// TIA Portal project "Ejercicio2" (V15.1)

(* hardware
DEVICE "HMI_1"  KTP700 Basic PN
   slot 0: "HMI_1"  KTP700 Basic PN  6AV2 123-2GB03-0AX0  15.1.0.0
   slot 1: "HMI_RT_1"  KTP700 Basic PN  6AV2 123-2GB03-0AX0  15.1.0.0
   slot 5: "HMI_1.IE_CP_1"  PROFINET Interface  15.0.1.0
      slot 1: "Interfaz PROFINET_1"  PROFINET Interface
         slot 1: "Port_1"  Port
DEVICE "S7-1200 station_1"  S7-1200 Station
   slot 0: "Rack_0"  S7-1200 Rack  Rack  V1.0
   slot 1: "PLC_1"  CPU 1215C AC/DC/Rly  6ES7 215-1BG40-0XB0  V4.2
*)

// ===== PLC "PLC_1"  CPU 1215C AC/DC/Rly =====

VAR_GLOBAL   // PLC tag table "Tabla de variables estándar"
   "System_Byte" AT %MB8191 : Byte;
   "FirstScan" AT %M8191.0 : Bool;
   "DiagStatusUpdate" AT %M8191.1 : Bool;
   "AlwaysTRUE" AT %M8191.2 : Bool;
   "AlwaysFALSE" AT %M8191.3 : Bool;
   "System_Byte(1)" AT %MB1 : Byte;
   "Clock_Byte" AT %MB100 : Byte;
   "Clock_10Hz" AT %M100.0 : Bool;
   "Clock_5Hz" AT %M100.1 : Bool;
   "Clock_2.5Hz" AT %M100.2 : Bool;
   "Clock_2Hz" AT %M100.3 : Bool;
   "Clock_1.25Hz" AT %M100.4 : Bool;
   "Clock_1Hz" AT %M100.5 : Bool;
   "Clock_0.625Hz" AT %M100.6 : Bool;
   "Clock_0.5Hz" AT %M100.7 : Bool;
   "Zona 1" AT %M0.0 : Bool;
   "Zona 2" AT %M0.1 : Bool;
   "Alarma ON/OFF" AT %M0.2 : Bool;
   "Alarma manual" AT %M0.3 : Bool;
   "LED sistema de alarma" AT %M10.0 : Bool;
   "Sirenea de alarma" AT %M10.1 : Bool;
   "Señal de alerta baja" AT %M10.2 : Bool;
   "Activar relé" AT %M10.3 : Bool;
   "Estado Alarma" AT %M1.0 : Bool;
   "Estado Sirena" AT %M1.1 : Bool;
END_VAR

// folder: System blocks/Program resources

DATA_BLOCK "Temporizador90s"   // DB1
{ S7_Optimized_Access := 'TRUE' }
AUTHOR : Simatic
FAMILY : IEC
NAME : IEC_TMR
VERSION : 1.0
// stored: InstanceOfName IEC_TIMER
"IEC_TIMER"
BEGIN
END_DATA_BLOCK

DATA_BLOCK "Temporizador60s"   // DB2
{ S7_Optimized_Access := 'TRUE' }
AUTHOR : Simatic
FAMILY : IEC
NAME : IEC_TMR
VERSION : 1.0
// stored: InstanceOfName IEC_TIMER
"IEC_TIMER"
BEGIN
END_DATA_BLOCK

// folder: (top level)

ORGANIZATION_BLOCK "Main"   // OB1, LAD, ProgramCycle
TITLE = "Main Program Sweep (Cycle)"
{ S7_Optimized_Access := 'TRUE' }
VERSION : 0.1
   VAR_INPUT
      Initial_Call : Bool;   // Initial call of this OB
      Remanence : Bool;   // =True, if remanent data are available
   END_VAR
   VAR_TEMP   // added for the SCL form of the ladder/FBD networks
      _w1 : Bool;
   END_VAR
BEGIN

REGION Network 1: Encendido si está activado y parpadeante desactivado si zonas 1 y 2 abiertas
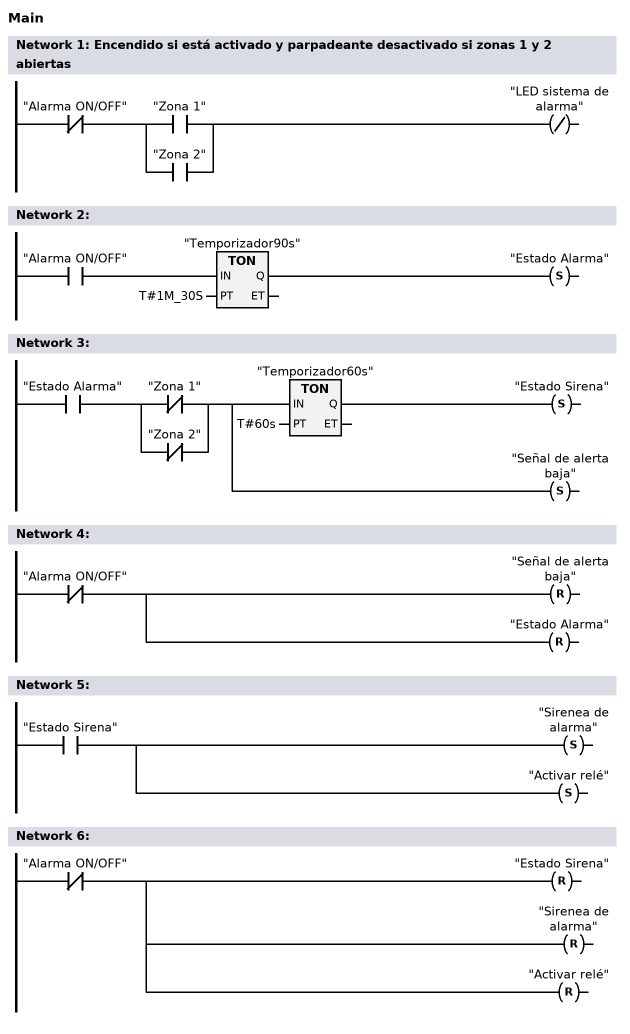
   RUNG wire#powerrail
      I_Contact( "Alarma ON/OFF" )
      wire#w1
      Contact( "Zona 1" )
      wire#w2
      I_Coil( "LED sistema de alarma" )
   END_RUNG
   RUNG wire#w1
      Contact( "Zona 2" )
   END_RUNG wire#w2
   // the same network as SCL:
   "LED sistema de alarma" := NOT (NOT "Alarma ON/OFF" AND ("Zona 1" OR "Zona 2"));
END_REGION

REGION Network 2
   "Temporizador90s".TON(IN := "Alarma ON/OFF", PT := T#1M_30S);
   IF "Temporizador90s".Q THEN "Estado Alarma" := TRUE; END_IF;
END_REGION

REGION Network 3
   #_w1 := "Estado Alarma" AND (NOT "Zona 1" OR NOT "Zona 2");
   "Temporizador60s".TON(IN := #_w1, PT := T#60s);
   IF "Temporizador60s".Q THEN "Estado Sirena" := TRUE; END_IF;
   IF #_w1 THEN "Señal de alerta baja" := TRUE; END_IF;
END_REGION

REGION Network 4
   RUNG wire#powerrail
      I_Contact( "Alarma ON/OFF" )
      wire#w1
      R_Coil( "Señal de alerta baja" )
   END_RUNG
   RUNG wire#w1
      R_Coil( "Estado Alarma" )
   END_RUNG
   // the same network as SCL:
   IF NOT "Alarma ON/OFF" THEN
       "Señal de alerta baja" := FALSE;
       "Estado Alarma" := FALSE;
   END_IF;
END_REGION

REGION Network 5
   RUNG wire#powerrail
      Contact( "Estado Sirena" )
      wire#w1
      S_Coil( "Sirenea de alarma" )
   END_RUNG
   RUNG wire#w1
      S_Coil( "Activar relé" )
   END_RUNG
   // the same network as SCL:
   IF "Estado Sirena" THEN
       "Sirenea de alarma" := TRUE;
       "Activar relé" := TRUE;
   END_IF;
END_REGION

REGION Network 6
   RUNG wire#powerrail
      I_Contact( "Alarma ON/OFF" )
      wire#w1
      R_Coil( "Estado Sirena" )
   END_RUNG
   RUNG wire#w1
      R_Coil( "Sirenea de alarma" )
   END_RUNG
   RUNG wire#w1
      R_Coil( "Activar relé" )
   END_RUNG
   // the same network as SCL:
   IF NOT "Alarma ON/OFF" THEN
       "Estado Sirena" := FALSE;
       "Sirenea de alarma" := FALSE;
       "Activar relé" := FALSE;
   END_IF;
END_REGION
END_ORGANIZATION_BLOCK

(* ===== HMI "HMI_RT_1" =====
system functions are stored by id; their names below are inferred from use
connection "HMI_Conexión_1": ETHERNET, SMART_S7_1200_OMS

HMI tags "Tabla de variables estándar"
   "Número_imagen_variable" : UInt, internal
   "Alarma ON/OFF" : Bool = PLC "Alarma ON/OFF" AT %M0.2, 1 s
   "Estado Alarma" : Bool = PLC "Estado Alarma" AT %M1.0, 1 s
   "Señal de alerta baja" : Bool = PLC "Señal de alerta baja" AT %M10.2, 1 s
   "Activar relé" : Bool = PLC "Activar relé" AT %M10.3, 1 s
   "LED sistema de alarma" : Bool = PLC "LED sistema de alarma" AT %M10.0, 1 s
   "Sirenea de alarma" : Bool = PLC "Sirenea de alarma" AT %M10.1, 1 s
   "Temporizador60s_ET" : Time = PLC Temporizador60s.ET, 1 s
   "Temporizador90s_ET" : Time = PLC Temporizador90s.ET, 1 s
   "Estado Sirena" : Bool = PLC "Estado Sirena" AT %M1.1, 1 s

text list "Nombre_imagen_lista_texto": 1 'Imagen raíz'

Template "Plantilla_1" 800x480
   Button "Salir" at 714,429 size 71x50; TextOff 'Salir'; PictureOff "ExitRuntime_KTP700_Basic_PN_TR"; PictureOn "ExitRuntime_KTP700_Basic_PN_TR"
      on Release: StopRuntime(0)
   Button "Template_Button" at 614,429 size 71x50; TextOff 'Text'
   Button "Template_Button_1" at 514,429 size 71x50; TextOff 'Text'
   Button "Template_Button_2" at 414,429 size 71x50; TextOff 'Text'
   Button "Template_Button_3" at 314,429 size 71x50; TextOff 'Text'
   Button "Template_Button_4" at 214,429 size 71x50; TextOff 'Text'
   Button "Template_Button_5" at 114,429 size 71x50; TextOff 'Text'
   Button "Imagen inicial" at 14,429 size 71x50; TextOff 'Imagen inicial'; PictureOff "NavigateHome_KTP700_Basic_PN_TR"; PictureOn "NavigateHome_KTP700_Basic_PN_TR"
      on Release: ActivateScreen("Imagen raíz", 0)
   SymbolicIOField "Imagen_campo_ES_simbólico" at 93,9 size 600x33; TextOff '0'; TextOn '1'; TextList "Nombre_imagen_lista_texto"
      ProcessValue <- "Número_imagen_variable"
      on Change: ActivateScreenByNumber("Número_imagen_variable", 0)
   DateTimeField "HmiScreenItemData" at 695,25 size 105x25
   DateTimeField "HmiScreenItemData_1" at 695,0 size 105x25
   GraphicView "Logotipo" at 0,0 size 91x51; Picture "Logotipo de HMI_1"

screen "Imagen raíz" 800x480, template "Plantilla_1"
   Switch "Interruptor_1" at 53,57 size 64x32; CaptionText 'Switch'; TextOff 'OFF'; TextOn 'ON'
      ProcessValue <- "Alarma ON/OFF"
   Circle "Círculo_1" at 247,52 size 48x48
      Appearance <- "Señal de alerta baja"
   Circle "Círculo_2" at 248,155 size 48x48
      Appearance <- "Activar relé"
   Circle "Círculo_3" at 247,222 size 48x48
      Appearance <- "Estado Sirena"
   Circle "Círculo_4" at 586,43 size 48x48
      Appearance <- "Alarma ON/OFF"
   TextField "Campo de texto_1" at 296,66 size 64x23; Text 'Alarma'
   TextField "Campo de texto_2" at 296,164 size 108x23; Text 'Aviso Policia'
   TextField "Campo de texto_3" at 296,233 size 57x23; Text 'Sirena'
   TextField "Campo de texto_4" at 642,57 size 158x23; Text 'Led estado Alarma'
   IOField "Campo ES_1" at 600,180 size 96x32; FormatPattern s9999999999
      ProcessValue <- "Temporizador60s_ET"
   IOField "Campo ES_2" at 599,272 size 96x32; FormatPattern s9999999999
      ProcessValue <- "Temporizador90s_ET"
*)